INTERFACE I_Sealer EXTENDS I_Module, I_TaskResult, I_Resettable, I_Override, I_ContainStatemachine

PROPERTY Recipe : REFERENCE TO ST_SealerRecipe
GET
END_GET
END_PROPERTY

PROPERTY SealBar : I_SealBar
GET
END_GET
END_PROPERTY

PROPERTY SealerAxis : I_Mc3Axis_PTP
GET
END_GET
END_PROPERTY

END_INTERFACE

(* stored: Version 1.1.0.1, ProductVersion 3.1.4026.20
   Itf I_Sealer: Id {374eec01-9f63-465f-96a9-4dee7b3bdec9}
   Property Recipe: Id {ecf572f4-816d-4883-87af-c52553c257d7}
   Get Get: Id {4ed5ed80-ef9f-4f46-a02c-5a59954dc9cd}
   Property SealBar: Id {4aab2e92-32ea-44b9-b581-f42fa3cb1a16}
   Get Get: Id {94805132-6838-422c-bc5a-41ebbc79109b}
   Property SealerAxis: Id {0552f28e-5fcb-44b6-bdd9-17ca7d619154}
   Get Get: Id {96dd9f9a-0002-4979-bff5-07599738a269} *)
